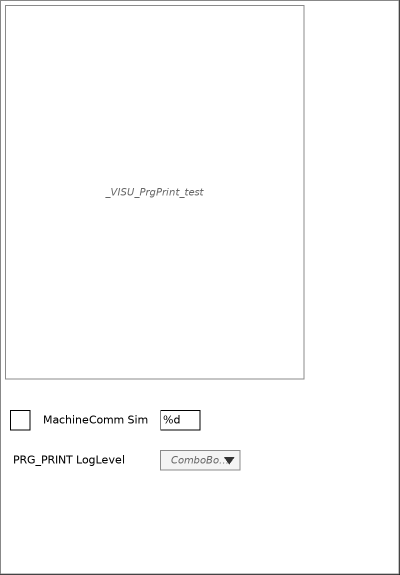
VISUALIZATION VIUS_TestnDebug  // 400x575
    Rectangle (0,0 400x575)
    Frame (5,5 299x374)
        shows _VISU_PrgPrint_test(mInst := PRG_PRINT.fbPrgPrintTest)
    Rectangle (160,410 40x20), "%d", tooltip "Simulation mode", text variable: PRG_MACHINE.fbMachineComm._nModeSel
        OnMouseClick: write the text variable via Default
    Rectangle (40,410 120x20), "MachineComm Sim"
    RoundedRectangle (10,410 20x20)
        toggle PRG_MACHINE.fbMachineComm.bSimEnable
    Rectangle (10,450 140x20), "PRG_PRINT LogLevel"
    ComboBoxInteger (160,450 80x20), tooltip "LogLevel", variable: PRG_PRINT.ePrint_LogLevel, text list: 'LogSeverity'
END_VISUALIZATION

(* stored: Version 1.1.0.1, ProductVersion 3.1.4024.11
   Visu VIUS_TestnDebug: Id {fc63999b-5a89-4067-8c94-8ec4b5f84340} *)
